Universal Robots PolyScope program: Project1pick6.urp

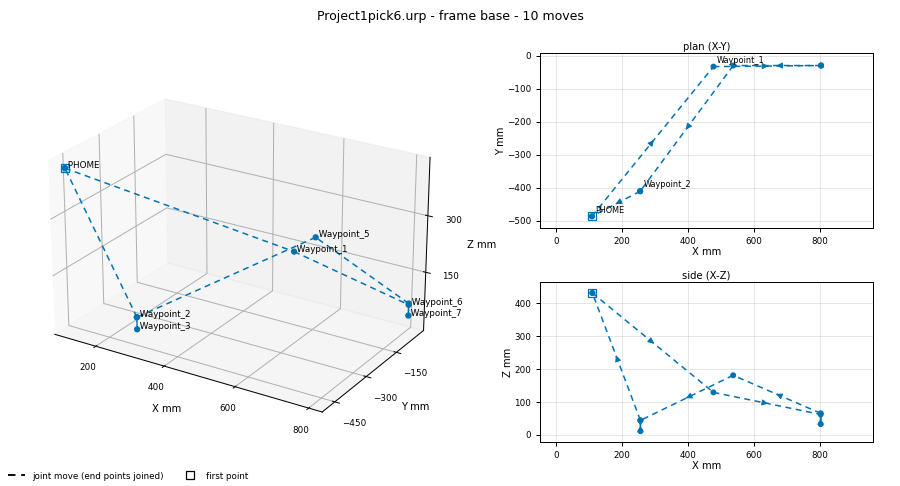
[picture p0: tool path of Project1pick6.urp in frame base, 10 of 10 moves have a stored position in this frame; points joined in program order, loops and branches not executed]
Program Project1pick6 (installation=admin directory=/programs/TUES_530PM createdIn=3.15.8.106339 lastSavedIn=3.15.8.106339 robotSerialNumber=2015350926)
Calibrated DH parameters: a=[0, -0.425, -0.39225, 0, 0, 0]; d=[0.089159, 0, 0, 0.10915, 0.09465, 0.0823]; alpha=[1.570796, 0, 0, 1.570796, -1.570796, 0]; deltaTheta=[0, 0, 0, 0, 0, 0]
Robot Program (runOnlyOnce=true)
  MoveJ speed 60 deg/s, acceleration 80 deg/s^2 (useActiveTCP=true)
    Waypoint PHOME: TCP in base x=109.127 y=-486.917 z=431.88 mm, rx=0.0001 ry=3.1416 rz=-0.0002 rad; joints [89.997, -90, 89.999, -90.006, -89.998, 0.001] deg
    Waypoint Waypoint_1: TCP in base x=477.218 y=-33.357 z=129.572 mm, rx=2.2261 ry=-2.212 rz=0.0055 rad; joints [162.86, -75.572, 123.035, -137.55, -90.266, -17.505] deg
    Waypoint Waypoint_6: TCP in base x=803.264 y=-30.051 z=62.587 mm, rx=2.2261 ry=-2.212 rz=0.0057 rad; joints [170.082, -33.741, 61.128, -117.446, -90.277, -10.281] deg
    Waypoint Waypoint_7: TCP in base x=803.244 y=-30.061 z=33.168 mm, rx=2.226 ry=-2.2118 rz=0.0054 rad; joints [170.081, -31.572, 61.598, -120.071, -90.28, -10.283] deg
    Wait Sleep waitTime=0.5
    Set DigitalOutput pin=digital_out[0]; digitalValue=1
    Wait Sleep waitTime=0.5
    Waypoint Waypoint_4: TCP in base x=803.272 y=-30.057 z=66.011 mm, rx=2.226 ry=-2.2119 rz=0.0055 rad; joints [170.082, -33.98, 61.044, -117.115, -90.281, -10.283] deg
    Waypoint Waypoint_5: TCP in base x=537.259 y=-30.095 z=181.531 mm, rx=2.2259 ry=-2.2118 rz=0.0054 rad; joints [165.134, -73.968, 110.575, -126.676, -90.279, -15.23] deg
    Waypoint Waypoint_2: TCP in base x=255.353 y=-410.745 z=44.444 mm, rx=-0.0208 ry=-3.1365 rz=-0.0002 rad; joints [108.873, -63.81, 124.974, -151.061, -90.272, 19.634] deg
    Waypoint Waypoint_3: TCP in base x=255.363 y=-410.797 z=11.544 mm, rx=-0.021 ry=-3.1365 rz=0.0001 rad; joints [108.872, -58.94, 125.262, -156.229, -90.273, 19.638] deg
    Wait Sleep waitTime=0.5
    Set DigitalOutput pin=digital_out[0]; digitalValue=0
    Wait Sleep waitTime=0.5
    Waypoint Waypoint_2: TCP in base x=255.353 y=-410.745 z=44.444 mm, rx=-0.0208 ry=-3.1365 rz=-0.0002 rad; joints [108.873, -63.81, 124.974, -151.061, -90.272, 19.634] deg
    Waypoint PHOME: TCP in base x=109.127 y=-486.917 z=431.88 mm, rx=0.0001 ry=3.1416 rz=-0.0002 rad; joints [89.997, -90, 89.999, -90.006, -89.998, 0.001] deg
